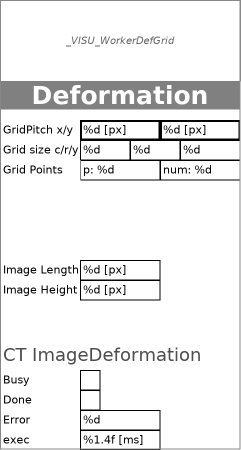
VISUALIZATION _VISU_WorkerDefGrid_Deformation  // 241x450
VAR_IN_OUT
		m_Inst : FB_WorkerDefGrid_Deformation;
END_VAR
    Rectangle (160,160 80x20), "num: %d", tooltip "num of grid points for job", text variable: m_Inst._sDeformationGridSettings.nGridPoints
    Rectangle (80,160 80x20), "p: %d", tooltip "processed grid points", text variable: m_Inst._nDeformationProcPoints[1]
    Frame (0,0 241x81)
        shows _VISU_WorkerDefGrid(m_Inst := m_Inst)
    Rectangle (0,120 160x20), "GridPitch x/y"
    Rectangle (160,120 80x20), "%d [px]", text variable: m_Inst._sDeformationGridSettings.nGridPitchY, input disabled if: m_Inst._pAttachedCt <> 0
        OnMouseDown: write the text variable via Default
    Rectangle (0,180 80x20)
    Rectangle (0,140 160x20), "Grid size c/r/y"
    Rectangle (130,140 50x20), "%d", tooltip "Grid SizeY", text variable: m_Inst._sDeformationGridSettings.nGridSizeY
    Label (0,340 240x30), "CT ImageDeformation"
    Rectangle (80,410 80x20), "%d", text variable: m_Inst._nDeformationErrorId, colour toggle: m_Inst._bDeformationError, invisible if: m_Inst._pAttachedCt = 0
    Rectangle (0,410 40x20), "Error"
    Rectangle (80,430 80x20), "%1.4f [ms]", text variable: m_Inst._tDeformationExecutionTime, invisible if: m_Inst._pAttachedCt = 0
    Rectangle (0,430 40x20), "exec"
    Rectangle (0,80 240x30), "Deformation", colour toggle: m_Inst._pAttachedCt <> 0
    Rectangle (80,120 80x20), "%d [px]", text variable: m_Inst._sDeformationGridSettings.nGridPitchX, input disabled if: m_Inst._pAttachedCt <> 0
        OnMouseDown: write the text variable via Default
    Rectangle (80,140 50x20), "%d", tooltip "Grid Size X", text variable: m_Inst._sDeformationGridSettings.nGridSizeX, input disabled if: m_Inst._pAttachedCt <> 0
        OnMouseDown: write the text variable via Default
    Rectangle (0,160 80x20), "Grid Points"
    Rectangle (0,370 80x20), "Busy"
    RoundedRectangle (80,370 20x20), colour toggle: m_Inst._bDeformationBusy, invisible if: m_Inst._pAttachedCt = 0, input disabled if: m_Inst._pAttachedCt <> 0
    Rectangle (0,390 80x20), "Done"
    RoundedRectangle (80,390 20x20), colour toggle: m_Inst._bDeformationDone, invisible if: m_Inst._pAttachedCt = 0
    Rectangle (0,260 80x20), "Image Length"
    Rectangle (0,280 80x20), "Image Height"
    Rectangle (80,260 80x20), "%d [px]", text variable: m_Inst._nImageDepthPx
    Rectangle (80,280 80x20), "%d [px]", text variable: m_Inst._nImageWidthPx
    Rectangle (180,140 60x20), "%d", tooltip "Grid ImageOffset Y [px]", text variable: m_Inst._sDeformationGridSettings.nGridImageOffsetY
END_VISUALIZATION

(* stored: Version 1.1.0.1, ProductVersion 3.1.4024.9
   Visu _VISU_WorkerDefGrid_Deformation: Id {e6c91e55-ff0b-4e93-a921-cff1a4b7baa0} *)
